FUNCTION FC_AnalogOutputValueHandling
VAR_INPUT
	Setpoint	:	REAL;
	UpperLimit	:	REAL;
	LowerLimit	:	REAL;
END_VAR
VAR_OUTPUT
	ConvertedValue	:	WORD;
END_VAR
VAR
	tempCalculatedValue	:	REAL;
	tempConvertedValue	:	WORD;
	tempValueWithOffset	:	WORD;
END_VAR

tempCalculatedValue := Setpoint * 10.0/(UpperLimit - LowerLimit);
tempConvertedValue := TO_WORD(tempCalculatedValue * 10.0);
tempValueWithOffset := tempConvertedValue * 10;

ConvertedValue := tempValueWithOffset;

END_FUNCTION

(* stored: Version 1.1.0.1
   POU FC_AnalogOutputValueHandling: Id {210ee896-c68b-4c74-929c-bd0f2c787fe8}, SpecialFunc None *)
